% RSLogix 500 project I2P JOB 15 - MYAH.RSS, saved by version 10.00.00.00 %
PROJECT "ML05B"    % processor: Bul.1763 MicroLogix 1100 Series B %

PROGRAM FILES
  LAD 2   16 rungs

DATA FILES
  O0 OUTPUT  4 elements
  I1 INPUT  6 elements
  S2 STATUS  66 elements
  B3 BINARY  1 elements
  T4 TIMER  1 elements
  C5 COUNTER  1 elements
  R6 CONTROL  1 elements
  N7 INTEGER  1 elements
  F8 FLOAT  1 elements

LADDER 2
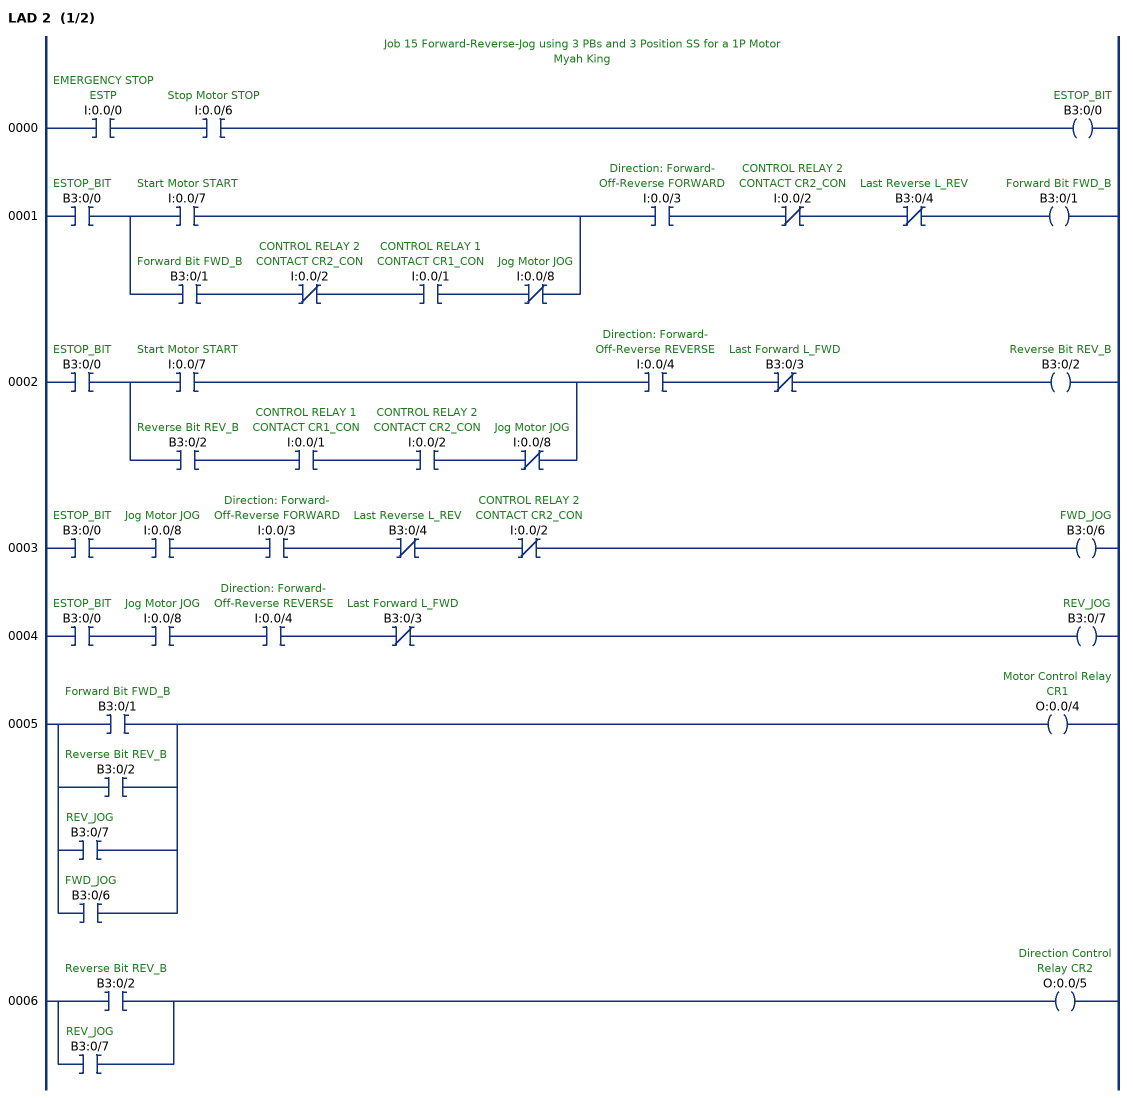
% Rung: 0 %
% Job 15 Forward-Reverse-Jog using 3 PBs and 3 Position SS for a 1P Motor
% Myah King %
SOR XIC I:0.0/0 XIC I:0.0/6 OTE B3:0/0 EOR
%   I:0.0/0  ESTP  "EMERGENCY STOP" %
%   I:0.0/6  STOP  "Stop Motor" %
%   B3:0/0  ESTOP_BIT %
% Rung: 1 %
SOR XIC B3:0/0 BST XIC I:0.0/7 NXB XIC B3:0/1 XIO I:0.0/2 XIC I:0.0/1 XIO I:0.0/8 BND XIC I:0.0/3 XIO I:0.0/2 XIO B3:0/4 OTE B3:0/1 EOR
%   B3:0/0  ESTOP_BIT %
%   I:0.0/7  START  "Start Motor" %
%   B3:0/1  FWD_B  "Forward Bit" %
%   I:0.0/2  CR2_CON  "CONTROL RELAY 2 CONTACT" %
%   I:0.0/1  CR1_CON  "CONTROL RELAY 1 CONTACT" %
%   I:0.0/8  JOG  "Jog Motor" %
%   I:0.0/3  FORWARD  "Direction: Forward- Off-Reverse" %
%   B3:0/4  L_REV  "Last Reverse" %
% Rung: 2 %
SOR XIC B3:0/0 BST XIC I:0.0/7 NXB XIC B3:0/2 XIC I:0.0/1 XIC I:0.0/2 XIO I:0.0/8 BND XIC I:0.0/4 XIO B3:0/3 OTE B3:0/2 EOR
%   B3:0/0  ESTOP_BIT %
%   I:0.0/7  START  "Start Motor" %
%   B3:0/2  REV_B  "Reverse Bit" %
%   I:0.0/1  CR1_CON  "CONTROL RELAY 1 CONTACT" %
%   I:0.0/2  CR2_CON  "CONTROL RELAY 2 CONTACT" %
%   I:0.0/8  JOG  "Jog Motor" %
%   I:0.0/4  REVERSE  "Direction: Forward- Off-Reverse" %
%   B3:0/3  L_FWD  "Last Forward" %
% Rung: 3 %
SOR XIC B3:0/0 XIC I:0.0/8 XIC I:0.0/3 XIO B3:0/4 XIO I:0.0/2 OTE B3:0/6 EOR
%   B3:0/0  ESTOP_BIT %
%   I:0.0/8  JOG  "Jog Motor" %
%   I:0.0/3  FORWARD  "Direction: Forward- Off-Reverse" %
%   B3:0/4  L_REV  "Last Reverse" %
%   I:0.0/2  CR2_CON  "CONTROL RELAY 2 CONTACT" %
%   B3:0/6  FWD_JOG %
% Rung: 4 %
SOR XIC B3:0/0 XIC I:0.0/8 XIC I:0.0/4 XIO B3:0/3 OTE B3:0/7 EOR
%   B3:0/0  ESTOP_BIT %
%   I:0.0/8  JOG  "Jog Motor" %
%   I:0.0/4  REVERSE  "Direction: Forward- Off-Reverse" %
%   B3:0/3  L_FWD  "Last Forward" %
%   B3:0/7  REV_JOG %
% Rung: 5 %
SOR BST XIC B3:0/1 NXB BST XIC B3:0/2 NXB BST XIC B3:0/7 NXB XIC B3:0/6 BND BND BND OTE O:0.0/4 EOR
%   B3:0/1  FWD_B  "Forward Bit" %
%   B3:0/2  REV_B  "Reverse Bit" %
%   B3:0/7  REV_JOG %
%   B3:0/6  FWD_JOG %
%   O:0.0/4  CR1  "Motor Control Relay" %
% Rung: 6 %
SOR BST XIC B3:0/2 NXB XIC B3:0/7 BND OTE O:0.0/5 EOR
%   B3:0/2  REV_B  "Reverse Bit" %
%   B3:0/7  REV_JOG %
%   O:0.0/5  CR2  "Direction Control Relay" %

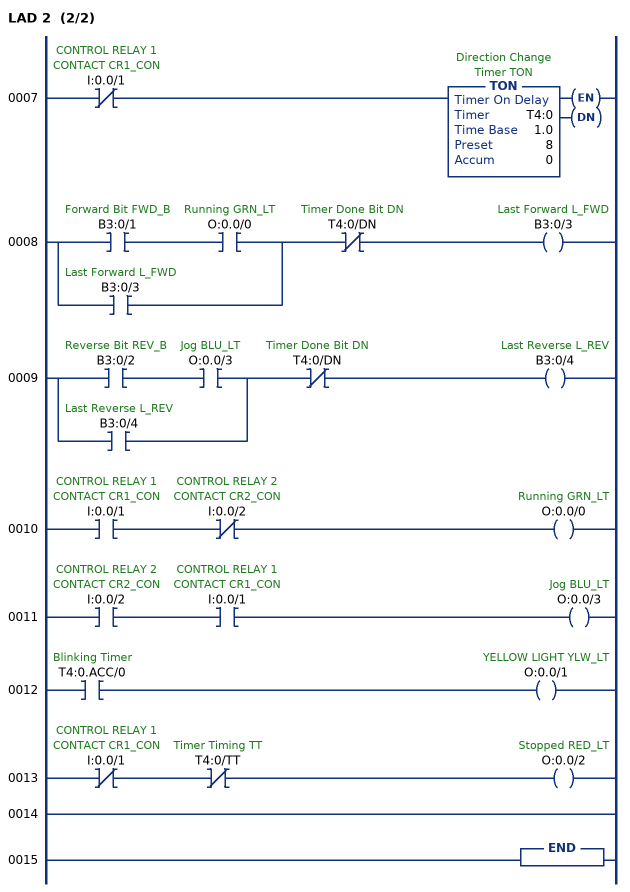
% Rung: 7 %
SOR XIO I:0.0/1 TON T4:0 1.0 8 0 EOR
%   I:0.0/1  CR1_CON  "CONTROL RELAY 1 CONTACT" %
%   T4:0  TON  "Direction Change Timer" %
% Rung: 8 %
SOR BST XIC B3:0/1 XIC O:0.0/0 NXB XIC B3:0/3 BND XIO T4:0/DN OTE B3:0/3 EOR
%   B3:0/1  FWD_B  "Forward Bit" %
%   O:0.0/0  GRN_LT  "Running" %
%   B3:0/3  L_FWD  "Last Forward" %
%   T4:0/DN  DN  "Timer Done Bit" %
% Rung: 9 %
SOR BST XIC B3:0/2 XIC O:0.0/3 NXB XIC B3:0/4 BND XIO T4:0/DN OTE B3:0/4 EOR
%   B3:0/2  REV_B  "Reverse Bit" %
%   O:0.0/3  BLU_LT  "Jog" %
%   B3:0/4  L_REV  "Last Reverse" %
%   T4:0/DN  DN  "Timer Done Bit" %
% Rung: 10 %
SOR XIC I:0.0/1 XIO I:0.0/2 OTE O:0.0/0 EOR
%   I:0.0/1  CR1_CON  "CONTROL RELAY 1 CONTACT" %
%   I:0.0/2  CR2_CON  "CONTROL RELAY 2 CONTACT" %
%   O:0.0/0  GRN_LT  "Running" %
% Rung: 11 %
SOR XIC I:0.0/2 XIC I:0.0/1 OTE O:0.0/3 EOR
%   I:0.0/2  CR2_CON  "CONTROL RELAY 2 CONTACT" %
%   I:0.0/1  CR1_CON  "CONTROL RELAY 1 CONTACT" %
%   O:0.0/3  BLU_LT  "Jog" %
% Rung: 12 %
SOR XIC T4:0.ACC/0 OTE O:0.0/1 EOR
%   T4:0.ACC/0  "Blinking Timer" %
%   O:0.0/1  YLW_LT  "YELLOW LIGHT" %
% Rung: 13 %
SOR XIO I:0.0/1 XIO T4:0/TT OTE O:0.0/2 EOR
%   I:0.0/1  CR1_CON  "CONTROL RELAY 1 CONTACT" %
%   T4:0/TT  TT  "Timer Timing" %
%   O:0.0/2  RED_LT  "Stopped" %
% Rung: 14 %  % edit flag set %
SOR EOR
% Rung: 15 %
SOR END EOR

OTHER DOCUMENTED ADDRESSES
  I:0.0/5  2PSS  "2 POSITION SELECTOR SWITCH"
  T4:0.ACC  BLINKING  "Timer Accumulater"

DATA TABLE (non-zero values as saved)
DATA B3
% B3:0 % 0X0001
DATA T4
% .PRE .ACC %
% T4:0 % 8 0
